// TIA Portal project "drill" (V18)

(* hardware
DEVICE "S7-1200-Station_1"  S7-1200 Station
   slot 0: "Baugruppenträger_0"  S7-1200 Rack  Rack  V1.0
   slot 1: "DRILL"  CPU 1215C DC/DC/DC  6ES7 215-1AG40-0XB0  V4.5
*)

// ===== PLC "DRILL"  CPU 1215C DC/DC/DC =====

VAR_GLOBAL   // PLC tag table "Standard-Variablentabelle"
   "eingang_LS" AT %I0.0 : Bool;
   "bearbeitung_LS" AT %I0.1 : Bool;
   "sauger_innen" AT %I0.2 : Bool;
   "sauger_außen" AT %I0.3 : Bool;
   "band_rein" AT %Q0.0 : Bool;
   "band_raus" AT %Q0.1 : Bool;
   "sauger_rein" AT %Q0.2 : Bool;
   "sauger_raus" AT %Q0.3 : Bool;
   "ventil_sauger_unten" AT %Q0.4 : Bool;
   "ventil_vakuum" AT %Q0.5 : Bool;
   "kompressor" AT %Q0.6 : Bool;
   "drill" AT %Q0.7 : Bool;
   "band_PWM" AT %Q1.0 : Bool;
   "sauger_PWM" AT %Q1.1 : Bool;
END_VAR

DATA_BLOCK "LOOP_DB"   // DB2
{ S7_Optimized_Access := 'TRUE' }
VERSION : 0.1
// stored: InstanceOfName LOOP
"LOOP"
BEGIN
END_DATA_BLOCK

FUNCTION_BLOCK "LOOP"   // FB1, SCL
{ S7_Optimized_Access := 'TRUE' }
VERSION : 0.1
   VAR
      warte : TON_TIME;
      warte_zeit : Time := T#500ms;
      warte_start : Bool;
      "step" : Int;
      pick : Bool;
      drop : Bool;
      drill : Bool;
      pick_finished : Bool;
      drop_finished : Bool;
      drill_finished : Bool;
      duration : Int := 2;
      idle : Bool;
   END_VAR
   VAR RETAIN
      model : String := 'DRILL';
   END_VAR
   VAR
      pick_failed : Bool;
      drop_failed : Bool;
      pick_aktiv : Bool;
      drop_aktiv : Bool;
      drill_aktiv : Bool;
   END_VAR
   VAR RETAIN
      zeit_prozessende : Time := T#2S;   // Zeit bevor die ProzessEnde Flag in der OPCUA-Schnittstelle gesetzt wird
      zeit_saugerRunter : Time := T#1000MS;   // Zeit die der Sauger nach unten gedrückt wird und dort verharrt
      zeit_vakuumLoesen : Time := T#500MS;   // Zeit die gewartet wird um dem Saugnapf die möglichkeit zu geben sich zu lösen
   END_VAR
   VAR
      "version" : String := '1.3.0';   // Version
   END_VAR
   VAR RETAIN
      zeit_vorFehlerchek : Time := T#2S;   // Zeit die vor dem Fehlercheck die nach dem PICK gewartet wird
      zeit_nachBohren : Time := T#500MS;   // Zeit die nach dem Bohren gewartet wird
      zeit_vakuumErzeugen : Time := T#200MS;   // Zeit für den Kompressor Vakuum aufzubauen
      zeit_mitteLS : Time := T#200MS;   // Zeit die das Band weiterfährt um das WP mittig in der Lichtschranke zu positionieren
   END_VAR
BEGIN
   #warte(IN := #warte_start,
               PT := #warte_zeit);

   // Stepchain MILL
        CASE #step OF
            0: // init
                #step := 1;
            1: // rdy
                #pick_finished := FALSE;
                #drop_finished := FALSE;
                #drill_finished := FALSE;
                #pick_failed := FALSE;
                #drop_failed := FALSE;
                #idle := TRUE;
                #step := 5;
            5: // Fallunterscheidung
                IF #pick THEN
                    #pick_aktiv := TRUE;
                    #pick := FALSE;
                    #idle := FALSE;
                    #step := 10;
                ELSIF #drop THEN
                    #drop_aktiv := TRUE;
                    #drop := FALSE;
                    #idle := FALSE;
                    #step := 100;
                ELSIF #drill THEN
                    #drill := FALSE;
                    #drill_aktiv := TRUE;
                    #idle := FALSE;
                    #step := 40;
                END_IF;
            200: // ENDE jedes Prozesses
                "band_PWM" := FALSE;
                "band_raus" := FALSE;
                "band_rein" := FALSE;
                "sauger_PWM" := FALSE;
                "sauger_raus" := FALSE;
                "sauger_rein" := FALSE;
                #warte_zeit := #zeit_prozessende;
                #warte_start := TRUE;
                IF #warte.Q THEN
                    #step := 1;
                    #warte_start := FALSE;
                END_IF
                ;

            10: // ----------------------------------------------------- START PICK
                // sauger raus bis schalter
                "sauger_PWM" := TRUE;
                "sauger_raus" := TRUE;
                IF "sauger_außen" THEN
                    "sauger_raus" := FALSE;
                    #step := 21;
                END_IF;

            21: // Sauger nimmt WP auf
                "kompressor" := TRUE;
                #step := 25;
            25: // warten Vakuum Erzeugung
                #warte_zeit := #zeit_vakuumErzeugen;
                #warte_start := TRUE;
                IF #warte.Q THEN
                    #warte_start := FALSE;
                    #step := 22;
                END_IF;
            22: // saugerkopf nach unten
                "ventil_sauger_unten" := TRUE;
                #warte_zeit := #zeit_saugerRunter;
                #warte_start := TRUE;
                IF #warte.Q THEN
                    #warte_start := FALSE;
                    #step := 23;
                END_IF;
            23: // Saugerkopf aktivieren
                "ventil_vakuum" := TRUE;
                #warte_zeit := #zeit_vakuumErzeugen;
                #warte_start := TRUE;
                IF #warte.Q THEN
                    #warte_start := FALSE;
                    #step := 24;
                END_IF;
            24: // saugerkopf nach oben
                "ventil_sauger_unten" := FALSE;
                #step := 30;
            30: // Sauger fährt rein
                "sauger_rein" := TRUE;
                IF "sauger_innen" THEN
                    "sauger_rein" := FALSE;
                    #step := 31;
                END_IF;
            31: // saugerkopf deaktivieren und runter
                "ventil_sauger_unten" := TRUE;
                #warte_zeit := #zeit_saugerRunter;
                #warte_start := TRUE;
                IF #warte.Q THEN
                    "ventil_vakuum" := FALSE;
                    #warte_start := FALSE;
                    #step := 32;
                END_IF;
            32: // Warten bis werkstück gelöst
                #warte_zeit := #zeit_vakuumLoesen;
                #warte_start := TRUE;
                IF #warte.Q THEN
                    "kompressor" := FALSE;
                    #warte_start := FALSE;
                    #step := 33;
                END_IF;
            33: // saugerkopf nach oben und aus
                "ventil_sauger_unten" := FALSE;
                #warte_zeit := #zeit_vorFehlerchek;
                #warte_start := TRUE;
                IF #warte.Q THEN
                    #warte_start := FALSE;
                    #step := 34;
                END_IF;
            34: // warten und fertig
                IF "eingang_LS" THEN // Fehlercheck
                    #pick_failed := TRUE;
                ELSE
                    #pick_finished := TRUE;
                END_IF;
                #pick_aktiv := FALSE;
                #step := 200;
                // ------------------------- ENDE PICK
            40: // ----------------------------------------------------- START DRILL
                // Power auf Band
                "band_PWM" := TRUE;
                #step := 41;
            41: // band rein wenn LS 
                "band_rein" := TRUE;
                IF NOT "bearbeitung_LS" THEN
                    #step := 42;
                END_IF;
            42: // Band laufen lassen bis mittig über drill
                #warte_zeit := #zeit_mitteLS;
                #warte_start := TRUE;
                IF #warte.Q THEN
                    "band_rein" := FALSE;
                    #warte_start := FALSE;
                    #step := 43;
                END_IF;
            43: // Bohren
                "drill" := TRUE;
                #warte_start := TRUE;
                #warte_zeit := T#1000ms * #duration;
                IF #warte.Q THEN
                    #warte_start := FALSE;
                    "drill" := FALSE;
                    #step := 44;
                END_IF;
            44: // warten nach bohren
                #warte_start := TRUE;
                #warte_zeit := #zeit_nachBohren;
                IF #warte.Q THEN
                    #warte_start := FALSE;
                    #step := 45;
                END_IF;
            45: // Band raus bis Eingang LS
                "band_raus" := TRUE;
                IF NOT "eingang_LS" THEN
                    #step := 46;
                END_IF;
            46: // Band weiter bis mittig unter sauger
                #warte_start := TRUE;
                #warte_zeit := #zeit_mitteLS;
                IF #warte.Q THEN
                    "band_raus" := FALSE;
                    #warte_start := FALSE;
                    #step := 50;
                END_IF;
            50: // drill finished
                #drill_aktiv := FALSE;
                #drill_finished := TRUE;
                #step := 200;
                // ------------------------- ENDE DRILL
            100:// ----------------------------------------------------- Start DROP
                // Power auf sauger und kompressor
                "kompressor" := TRUE;
                "sauger_PWM" := TRUE;
                #step := 120;
            120: // Sauger fährt rein
                "sauger_rein" := TRUE;
                IF "sauger_innen" THEN
                    "sauger_rein" := FALSE;
                    #step := 101;
                END_IF;
            101: // saugerkopf nach unten
                "ventil_sauger_unten" := TRUE;
                #step := 102;
            102: // Saugerkopf aktivieren
                #warte_zeit := #zeit_saugerRunter;
                #warte_start := TRUE;
                IF #warte.Q THEN
                    "ventil_vakuum" := TRUE;
                    #warte_start := FALSE;
                    #step := 103;
                END_IF;
            103: // saugerkopf nach oben
                #warte_zeit := #zeit_vakuumErzeugen;
                #warte_start := TRUE;
                IF #warte.Q THEN
                    #warte_start := FALSE;
                    "ventil_sauger_unten" := FALSE;
                    #step := 104;
                END_IF
                ;
            104: // sauger raus bis schalter
                "sauger_raus" := TRUE;
                IF "sauger_außen" THEN
                    "sauger_raus" := FALSE;
                    #step := 105;
                END_IF;
            105: // saugerkopf nach unten
                "ventil_sauger_unten" := TRUE;
                #step := 106;
            106: // saugerkopf deaktivieren
                #warte_start := TRUE;
                #warte_zeit := #zeit_saugerRunter;
                IF #warte.Q THEN
                    "ventil_vakuum" := FALSE;
                    #warte_start := FALSE;
                    #step := 107;
                END_IF;
            107: // Warten bis werkstück sich löst
                #warte_start := TRUE;
                #warte_zeit := #zeit_vakuumLoesen;
                IF #warte.Q THEN
                    #warte_start := FALSE;
                    #step := 108;
                END_IF;
            108: // saugerkopf nach oben und kompressor aus
                "kompressor" := FALSE;
                #warte_start := TRUE;
                #warte_zeit := T#300ms;
                IF #warte.Q THEN
                    "ventil_sauger_unten" := FALSE;
                    #warte_start := FALSE;
                    #step := 109;
                END_IF;
            109: // warten
                #warte_start := TRUE;
                #warte_zeit := #zeit_vakuumLoesen;
                IF #warte.Q THEN
                    #warte_start := FALSE;
                    #step := 110;
                END_IF;
            110: // reinfahren
                "sauger_rein" := TRUE;
                IF "sauger_innen" THEN
                    "sauger_rein" := FALSE;
                    #step := 112;
                END_IF;
            112: // drop reset 
                IF NOT "eingang_LS" THEN
                    #drop_failed := TRUE;
                ELSE
                    #drop_finished := TRUE;
                END_IF;
                #drop_aktiv := FALSE;
                #step := 200;
                // ------------------------- ENDE DROP
            ELSE
                ;
        END_CASE;
END_FUNCTION_BLOCK

ORGANIZATION_BLOCK "Main"   // OB1, LAD, ProgramCycle
TITLE = "Main Program Sweep (Cycle)"
{ S7_Optimized_Access := 'TRUE' }
VERSION : 0.1
   VAR_INPUT
      Initial_Call : Bool;   // Initial call of this OB
      Remanence : Bool;   // =True, if remanent data are available
   END_VAR
BEGIN

REGION Network 1
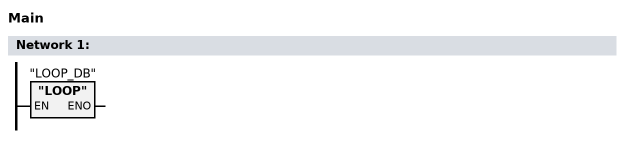
   RUNG wire#powerrail
      "LOOP_DB"()
   END_RUNG
   // the same network as SCL:
   "LOOP_DB"();   // "LOOP"
END_REGION
END_ORGANIZATION_BLOCK